INTERFACE itfCommand

METHOD Abort : MC_Error
VAR_INPUT
END_VAR
END_METHOD

PROPERTY Active : BOOL
GET
END_GET
END_PROPERTY

PROPERTY Busy : BOOL
GET
END_GET
END_PROPERTY

PROPERTY Command : MC_COMMAND_REF
GET
END_GET
END_PROPERTY

PROPERTY CommandAborted : BOOL
GET
END_GET
END_PROPERTY

PROPERTY Done : BOOL
GET
END_GET
END_PROPERTY

PROPERTY Error : BOOL
GET
END_GET
END_PROPERTY

PROPERTY ErrorId : UDINT
GET
END_GET
END_PROPERTY

METHOD Wait : MC_Error // This method only makes sense in the IEC 61499 environment
VAR_INPUT
	Timeout : TIME;
	AbortOnTimeout : BOOL; 
END_VAR
END_METHOD

END_INTERFACE

(* stored: Version 1.1.0.1, ProductVersion 3.1.4024.12
   Itf itfCommand: Id {7dbdb552-aff2-43fc-95ff-b80cdb7109a5}
   Method Abort: Id {71cb0fe7-f024-469d-a609-416dab4b5cdf}
   Property Active: Id {864b292b-df5a-420f-9462-8b7e67645ce3}
   Get Get: Id {19609267-cbf8-4722-b1bf-6d62c7303c99}
   Property Busy: Id {5ac40040-df89-41c2-af36-124994a82c04}
   Get Get: Id {169f8eb3-de93-4c3c-8b30-edd673640ca5}
   Property Command: Id {409ab707-8363-4fa5-93f9-cd50f90dd4dd}
   Get Get: Id {af3de311-2054-4e97-b9e2-5a456a006dcd}
   Property CommandAborted: Id {84c7d780-28c4-465a-86c8-063de9e042a6}
   Get Get: Id {8d5c7a8f-3d5d-4056-93c4-0d2a6b58a3b6}
   Property Done: Id {dc85e9d5-6d70-4957-b9a8-ac3b4dbd02d7}
   Get Get: Id {d68b9c8f-823f-4c62-838a-0570d9da8db5}
   Property Error: Id {5c194584-797d-4b52-bc0f-89b53dc6ae26}
   Get Get: Id {1ea88778-0737-4551-8457-a20a9e1cdb2e}
   Property ErrorId: Id {5c077f40-b3c9-4eb8-9ab7-e2bfcf3410a2}
   Get Get: Id {fb7a1a80-52d6-41b6-b23b-a7702ed89244}
   Method Wait: Id {7bb16dc8-dced-422b-8d79-d1f6b6d9da19} *)
